// Mitsubishi GX Works2 project: 동작요구동작   PLC: Q02/Q02H

PROGRAM MAIN
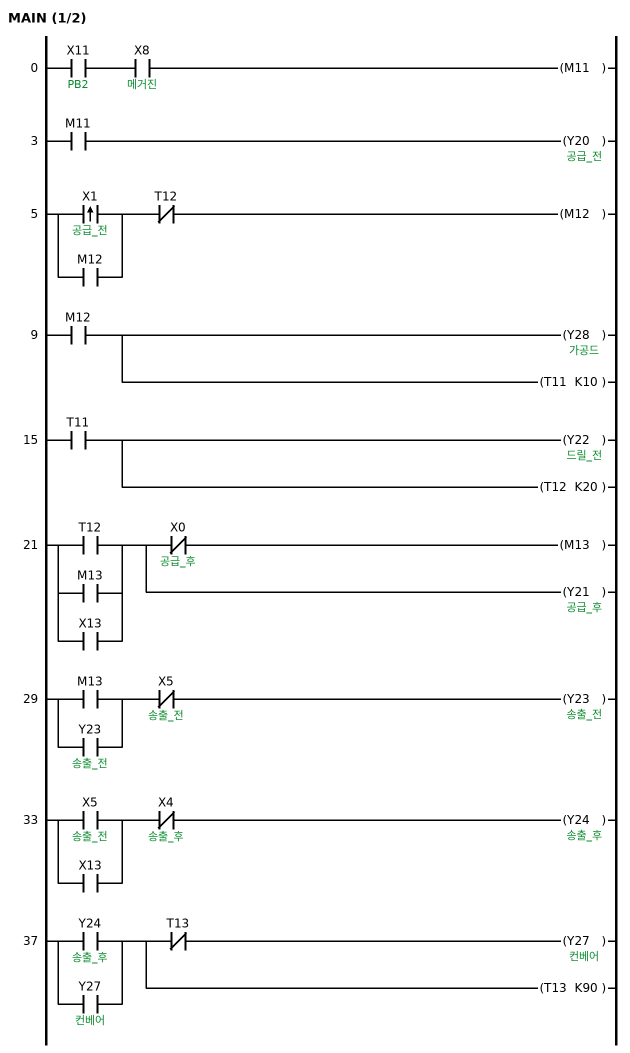
0     LD      X11  ; PB2
      AND     X8  ; 메거진
      OUT     M11
3     LD      M11
      OUT     Y20  ; 공급_전
5     LDP     X1  ; 공급_전
      OR      M12
      ANI     T12
      OUT     M12
9     LD      M12
      OUT     Y28  ; 가공드
      OUT     T11 K10
15    LD      T11
      OUT     Y22  ; 드릴_전
      OUT     T12 K20
21    LD      T12
      OR      M13
      OR      X13
      MPS
      ANI     X0  ; 공급_후
      OUT     M13
      MPP
      OUT     Y21  ; 공급_후
29    LD      M13
      OR      Y23  ; 송출_전
      ANI     X5  ; 송출_전
      OUT     Y23  ; 송출_전
33    LD      X5  ; 송출_전
      OR      X13
      ANI     X4  ; 송출_후
      OUT     Y24  ; 송출_후
37    LD      Y24  ; 송출_후
      OR      Y27  ; 컨베어
      MPS
      ANI     T13
      OUT     Y27  ; 컨베어
      MPP
      OUT     T13 K90
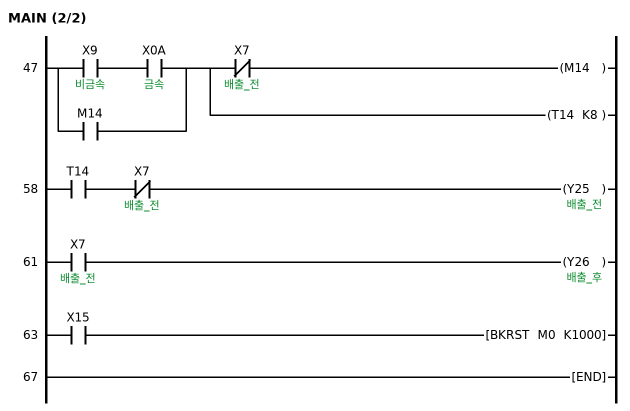
47    LD      X9  ; 비금속
      AND     X0A  ; 금속
      OR      M14
      MPS
      ANI     X7  ; 배출_전
      OUT     M14
      MPP
      OUT     T14 K8
58    LD      T14
      ANI     X7  ; 배출_전
      OUT     Y25  ; 배출_전
61    LD      X7  ; 배출_전
      OUT     Y26  ; 배출_후
63    LD      X15
      BKRST   M0 K1000
67    END
END_PROGRAM

// device comments not shown above
X2  ; 드릴_상
X3  ; 드릴_하
X6  ; 배출_후
X10  ; PB1
X12  ; PB3
Y29  ; 적색
Y2A  ; 황색
Y2B  ; 녹색
